TYPE T_SaveSlot : UINT(1..65535); END_TYPE

(* stored: Version 1.1.0.1, ProductVersion 3.1.4019.2
   DUT T_SaveSlot: Id {06cf4727-1aaf-48f4-9aeb-c9375eb66aaa} *)
